TYPE ST_Param :
STRUCT
  fValue    : LREAL;
  bValid    : BOOL;
  bWriteToNc  : BOOL;
END_STRUCT
END_TYPE

(* stored: Version 1.1.0.1, ProductVersion 3.1.4023.8
   DUT ST_Param: Id {c1fc51ab-8062-4d2a-b281-a05ced5079c0} *)
